# B&R Automation Studio project Ampel
Automation Studio 6.0.2.177; technology packages: OpcUaCs 6.0.0, OpcUaFx 6.0.0


## Logical view

### Program Logical/Ampel (ANSIC)

#### Variables.var
```iecst
VAR
	DurationGreenBlinking : USINT;
	DurationGreen : USINT;
	DurationYellow : USINT;
	DurationRed : USINT;
	LightYellow : BOOL;
	LightRed : BOOL;
	LightGreen : BOOL;
	CyclesCount : USINT;
	TraceMessages : ARRAY[0..200] OF STRING[80];
	CountDown : USINT;
END_VAR
```

#### States.hpp
```cpp
#include "machine.hpp"

// data shared between FSM states and outside code
struct Context {
	unsigned cycleCount = 0;
	unsigned countGreenBlinking = 0;
	unsigned countGreen = 0;
	unsigned countYellow = 0;
	unsigned countRed = 0;
};

// convenience typedef
using M = hfsm2::MachineT<hfsm2::Config::ContextT<Context>>;

// macro magic invoked to simplify FSM structure declaration
#define S(s) struct s

// State machine structure
using FSM = M::PeerRoot<
	// sub-machine ..
	M::Composite<S(On),
	// .. with 5 sub-states
	S(Red),
	S(YellowDownwards),
	S(YellowUpwards),
	S(GreenBlinking),
	S(Green)
	>,
				S(Off)
			>;
#undef S

//------------------------------------------------------------------------------

static_assert(FSM::regionId<On>()			  ==  1, "");

static_assert(FSM::stateId<On>()			  ==  1, "");
static_assert(FSM::stateId<Red>()			  ==  2, "");
static_assert(FSM::stateId<YellowDownwards>() ==  3, "");
static_assert(FSM::stateId<YellowUpwards>()	  ==  4, "");
static_assert(FSM::stateId<GreenBlinking>()	  ==  5, "");
static_assert(FSM::stateId<Green>()			  ==  6, "");
static_assert(FSM::stateId<Off>()			  ==  7, "");

////////////////////////////////////////////////////////////////////////////////

// top-level region in the hierarchy
struct On
	: FSM::State // necessary boilerplate!
{
	// called on state entry
	void enter(Control& control) {
		control.context().cycleCount = 0;
		TraceMessage("On");
	}
};

//------------------------------------------------------------------------------

// sub-states
struct Red
	: FSM::State
{
	void enter(Control& control) {
		++control.context().cycleCount;
		LightRed = true;
		LightYellow = false;
		LightGreen = false;
		control.context().countRed = 0;
		CountDown = DurationRed + DurationYellow + 2;
		TraceMessage("Red");

	}

	// state can initiate transitions to _any_ other state
	void update(FullControl& control) {

		// multiple transitions can be initiated, can be useful in a hierarchy
		if (control.context().cycleCount > 10)
			control.changeTo<Off>();
		else {
			if (control.context().countRed++ >= DurationRed){
				control.changeTo<YellowDownwards>();
			}
		}
		CountDown--;
	}
};

// - - - - - - - - - - - - - - - - - - - - - - - - - - - - - - - - - - - - - - -

struct YellowDownwards
	: FSM::State
{
	void enter(Control& control) {
		TraceMessage("Yellow v");
		LightYellow = true; //Keep Red On
		control.context().countYellow = 0;
	}

	void update(FullControl& control) {
		if (control.context().countYellow++ > DurationYellow) { //was 3
			control.changeTo<Green>();
		}
		CountDown--;
	}
};

// - - - - - - - - - - - - - - - - - - - - - - - - - - - - - - - - - - - - - - -

struct YellowUpwards
	: FSM::State
{
	void enter(Control& control) {
		TraceMessage("Yellow ^");
		LightGreen = false;
		LightYellow = true;
		control.context().countYellow = 0;
	}

	void update(FullControl& control) {
		if (control.context().countYellow++ > DurationYellow) {
			control.changeTo<Red>();
		}
	}
};

// - - - - - - - - - - - - - - - - - - - - - - - - - - - - - - - - - - - - - - -

struct GreenBlinking
	: FSM::State
{
	void enter(Control& control) {
		TraceMessage("Green Blinking");
		control.context().countGreenBlinking = 0;
	}

	void update(FullControl& control) {
		LightGreen = !LightGreen; // Blinking
		if ((control.context().countGreenBlinking++ > DurationGreenBlinking) && !LightGreen) {
			control.changeTo<YellowUpwards>();
		}
		CountDown--;
	}
};

// - - - - - - - - - - - - - - - - - - - - - - - - - - - - - - - - - - - - - - -

struct Green
	: FSM::State
{
	void enter(Control& control) {
		TraceMessage("Green");
		control.context().countGreen = 0;
		LightRed = false;
		LightYellow = false;
		LightGreen = true;
		CountDown = DurationGreen + DurationGreenBlinking + 4;
	}

	void update(FullControl& control) {
		if (control.context().countGreen++ > DurationGreen){
			control.changeTo<GreenBlinking>();
		}
		CountDown--;
	}
};

//------------------------------------------------------------------------------

// another top-level state
struct Off
	: FSM::State
{
	void enter(Control&) {
		TraceMessage("Off");
	}
};
```

#### Main.cpp
```cpp
#include <bur/plctypes.h>

#ifdef _DEFAULT_INCLUDES
	#include <AsDefault.h>
#endif

// amount of memory to be allocated for heap storage must be specified
// for every ANSI C++ program with the bur_heap_size variable
unsigned long bur_heap_size = 0xFFFF;

#include "machine.hpp"
#include "Logging.hpp"
#include "States.hpp"

////////////////////////////////////////////////////////////////////////////////

// shared data storage instance
Context context;
FSM::Instance machine{context};

void _INIT ProgramInit(void)
{
	// Insert code here
	CyclesCount = 0;
	ClearTraceLog();
	DurationRed = 5;
	DurationYellow = 3;
	DurationGreen = 5;
	DurationGreenBlinking = 3;
	LightRed = false;
	LightYellow = false;
	LightGreen = false;
}

void _CYCLIC ProgramCyclic(void)
{
	// Insert code here
	machine.update();
	CyclesCount++;
	TraceMessage("---cycle---");
}

void _EXIT ProgramExit(void)
{
	// Insert code here
}
```

Listed in the project but not available here: Logical/Global.typ, Logical/Global.var, Logical/Libraries
